FUNCTION_BLOCK E_T_FF
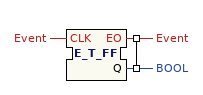
  EVENT_INPUT
    CLK;
  END_EVENT
  EVENT_OUTPUT
    EO WITH Q;
  END_EVENT
  VAR_OUTPUT
    Q : BOOL;
  END_VAR
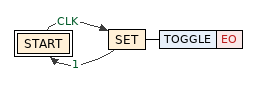
  EC_STATES
    START;
    SET : TOGGLE -> EO;
  END_STATES
  EC_TRANSITIONS
    START TO SET := CLK;
    SET TO START := 1;
  END_TRANSITIONS
  ALGORITHM TOGGLE IN ST:
Q := NOT Q;&#38;#10;
  END_ALGORITHM
END_FUNCTION_BLOCK
